Fanuc KAREL source: kb00011.KL

-- PROVISIONAL review KL for V1013-1; original PC SHA256 2ab2a836d27b45b5e5a6bb54155bc9eb2025235f9a95d708748d673243d2d142
-- Incomplete behavior may be omitted. Consult companion uncertainty JSON. Do not deploy.
PROGRAM KB00011
%NOLOCKGROUP
BEGIN
  -- UNRESOLVED_PC offsets 5-14; opcodes 3F,75
  -- UNRESOLVED_PC offsets 19-28; opcodes 3F,75
  -- UNRESOLVED_PC offsets 33-40; opcodes 9D,23
  -- UNRESOLVED_PC offsets 45-52; opcodes 9D,23
  -- UNRESOLVED_PC offsets 57-64; opcodes 9D,23
  -- UNRESOLVED_PC offsets 69-107; opcodes 27,22,2A,22,2A,22,22,22,31
  -- UNRESOLVED_PC offsets 112-116; opcodes 7F
END KB00011
